# EPICS autosave request: iocBoot/iocddrive/auto_settings.req
file motor_settings.req P=MLL:ddrive:,M=m1
